FUNCTION_BLOCK FB_TrackBase


VAR
	trackLinePosStart 	: PositionXYC;
	trackLinePosEnd 	: PositionXYC;
	fbTrackStandard		: FB_TrackStandard;
	fTrackLength		: LREAL;

	nState				: INT;
	sErrorInfoText		: STRING;
	sErrorInfoTextTemp	: STRING;
	bTrackBuildError	: BOOL;

END_VAR

METHOD Clear : BOOL


VAR_INST
	
	nStateReset		: UINT;

END_VAR


	CASE nStateReset OF
		
	0:	nStateReset := 10;
	
	10: IF fbTrackStandard.P_State = MC_PLANAR_STATE.Error
		OR fbTrackStandard.P_State = MC_PLANAR_STATE.ErrorPending
		THEN
			nStateReset := nStateReset +1;
		ELSE
			nStateReset := nStateReset +10;
		END_IF
		
	11: IF fbTrackStandard.Reset() THEN
			nStateReset := nStateReset +1;
		END_IF
	
	12:	IF fbTrackStandard.P_Reset.Done THEN
			nStateReset := nStateReset +8;
		END_IF
	
	20:
		  sErrorInfoText := '';
		bTrackBuildError := FALSE;
				  nState := 10;
				   Clear := TRUE;	
	
		nStateReset := 0;
	
	END_CASE
END_METHOD

METHOD Cycle : BOOL
VAR_INPUT
END_VAR
fbTrackStandard.Cycle();
END_METHOD

PROPERTY P_TrackLength : LREAL
GET
P_TrackLength := fTrackLength;
END_GET
END_PROPERTY

PROPERTY std : I_TrackStandard
GET
std := fbTrackStandard;
END_GET
END_PROPERTY

END_FUNCTION_BLOCK

(* stored: Version 1.1.0.1, ProductVersion 3.1.4024.9
   POU FB_TrackBase: Id {45178168-0bcd-4ee5-9303-985a149ae50d}, SpecialFunc None
   Method Clear: Id {2e12ce18-c1cf-4db0-8e6f-3cfa6f0b0586}
   Method Cycle: Id {6d99c307-83b1-4b38-bfc8-d359a388721a}
   Property P_TrackLength: Id {ae4ae5a2-da3b-4c87-9d92-ee3a7446bcff}
   Get Get: Id {aaef772e-37c7-44c0-8593-2daa4f5c1ab4}
   Property std: Id {2f5b9d63-b860-4bba-be2a-ce4713215f97}
   Get Get: Id {82bff7dd-b450-40b9-b243-d7324ca4a33a} *)
